(* IEC 61131-3 sources: plc-workspace/projects/FB_MainSequence/05_tia_sync/exported_scl, 6 files *)

(* ---- FC_MainSequence_BusyPhase.st ---- *)
FUNCTION FC_MainSequence_BusyPhase : BOOL
VAR_INPUT
    iPhase : INT := 0;
END_VAR

FC_MainSequence_BusyPhase := (iPhase = 1) OR (iPhase = 2) OR (iPhase = 3);

END_FUNCTION

(* ---- FC_MainSequence_InvalidPhase.st ---- *)
FUNCTION FC_MainSequence_InvalidPhase : BOOL
VAR_INPUT
    iPhase : INT := 0;
END_VAR

FC_MainSequence_InvalidPhase := (iPhase < 0) OR ((iPhase > 3) AND (iPhase <> 900));

END_FUNCTION

(* ---- FC_MainSequence_NextTimer.st ---- *)
FUNCTION FC_MainSequence_NextTimer : UINT
VAR_INPUT
    xResetReq : BOOL := FALSE;
    iPhaseStat : INT := 0;
    xInvalidPhase : BOOL := FALSE;
    xStepDone : BOOL := FALSE;
    xTimeoutReached : BOOL := FALSE;
    xBusyPhase : BOOL := FALSE;
    uiStepTimerStat : UINT := 0;
    uiStepTimeoutScans : UINT := 0;
END_VAR

IF xResetReq OR (iPhaseStat = 0) OR (iPhaseStat = 900) OR xInvalidPhase OR xStepDone OR xTimeoutReached THEN
    FC_MainSequence_NextTimer := 0;
ELSIF xBusyPhase AND (uiStepTimeoutScans > 0) THEN
    FC_MainSequence_NextTimer := uiStepTimerStat + 1;
ELSE
    FC_MainSequence_NextTimer := 0;
END_IF;

END_FUNCTION

(* ---- FC_MainSequence_StepDone.st ---- *)
FUNCTION FC_MainSequence_StepDone : BOOL
VAR_INPUT
    iPhase : INT := 0;
    xTransportDone : BOOL := FALSE;
    xFlipDone : BOOL := FALSE;
    xOutputDone : BOOL := FALSE;
END_VAR

CASE iPhase OF
    1:
        FC_MainSequence_StepDone := xTransportDone;
    2:
        FC_MainSequence_StepDone := xFlipDone;
    3:
        FC_MainSequence_StepDone := xOutputDone;
    ELSE
        FC_MainSequence_StepDone := FALSE;
END_CASE;

END_FUNCTION

(* ---- FC_MainSequence_SuccessPhase.st ---- *)
FUNCTION FC_MainSequence_SuccessPhase : INT
VAR_INPUT
    iPhase : INT := 0;
END_VAR

CASE iPhase OF
    1:
        FC_MainSequence_SuccessPhase := 2;
    2:
        FC_MainSequence_SuccessPhase := 3;
    3:
        FC_MainSequence_SuccessPhase := 1;
    ELSE
        FC_MainSequence_SuccessPhase := iPhase;
END_CASE;

END_FUNCTION

(* ---- FC_MainSequence_TimeoutReached.st ---- *)
FUNCTION FC_MainSequence_TimeoutReached : BOOL
VAR_INPUT
    xBusyPhase : BOOL := FALSE;
    xStepDone : BOOL := FALSE;
    uiStepTimerStat : UINT := 0;
    uiStepTimeoutScans : UINT := 0;
END_VAR

FC_MainSequence_TimeoutReached :=
    xBusyPhase AND
    (NOT xStepDone) AND
    (uiStepTimeoutScans > 0) AND
    ((uiStepTimerStat + 1) >= uiStepTimeoutScans);

END_FUNCTION
